// TIA Portal V20 export
TYPE "typeEm0Monitoring"
// stored: Access Published, Namespace Unit1
   STRUCT
      jobinterface { ExternalWritable := 'False'} : "Unit1.typeEm0MonitoringJobInterface";
      cmStatus { ExternalWritable := 'False'} : "Unit1.typeEm0MonitoringCmStatus";
      UserDefine { ExternalWritable := 'False'} : "Unit1.typeEm0MonitoringUserDefine";
   END_STRUCT;
END_TYPE
